% RSLogix 500 project P1.RSS, saved by version 8.10.00.18 %
PROJECT "UNTITLED"    % processor: MicroLogix 1200 %

PROGRAM FILES
  LAD 2 "MAIN"  3 rungs
  LAD 3 "IOS"  5 rungs
  LAD 4 "CONTROL"  11 rungs

DATA FILES
  O0 OUTPUT  4 elements
  I1 INPUT  4 elements
  S2 STATUS  66 elements
  B3 BINARY  1 elements
  T4 TIMER  4 elements
  C5 COUNTER  1 elements
  R6 CONTROL  1 elements
  N7 INTEGER  1 elements

LADDER 2 "MAIN"
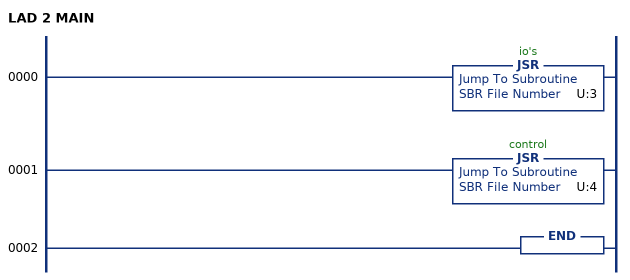
% Rung: 0 %
SOR JSR U:3 EOR
%   U:3  "io's" %
% Rung: 1 %
SOR JSR U:4 EOR
%   U:4  "control" %
% Rung: 2 %
SOR END EOR

LADDER 3 "IOS"
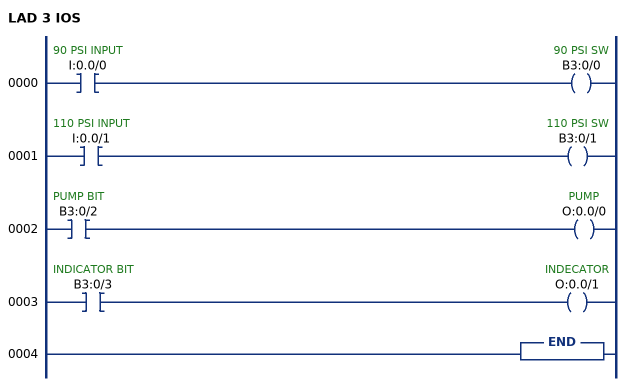
% Rung: 0 %
SOR XIC I:0.0/0 OTE B3:0/0 EOR
%   I:0.0/0  "90 PSI INPUT" %
%   B3:0/0  "90 PSI SW" %
% Rung: 1 %
SOR XIC I:0.0/1 OTE B3:0/1 EOR
%   I:0.0/1  "110 PSI INPUT" %
%   B3:0/1  "110 PSI SW" %
% Rung: 2 %
SOR XIC B3:0/2 OTE O:0.0/0 EOR
%   B3:0/2  "PUMP BIT" %
%   O:0.0/0  "PUMP" %
% Rung: 3 %
SOR XIC B3:0/3 OTE O:0.0/1 EOR
%   B3:0/3  "INDICATOR BIT" %
%   O:0.0/1  "INDECATOR" %
% Rung: 4 %
SOR END EOR

LADDER 4 "CONTROL"
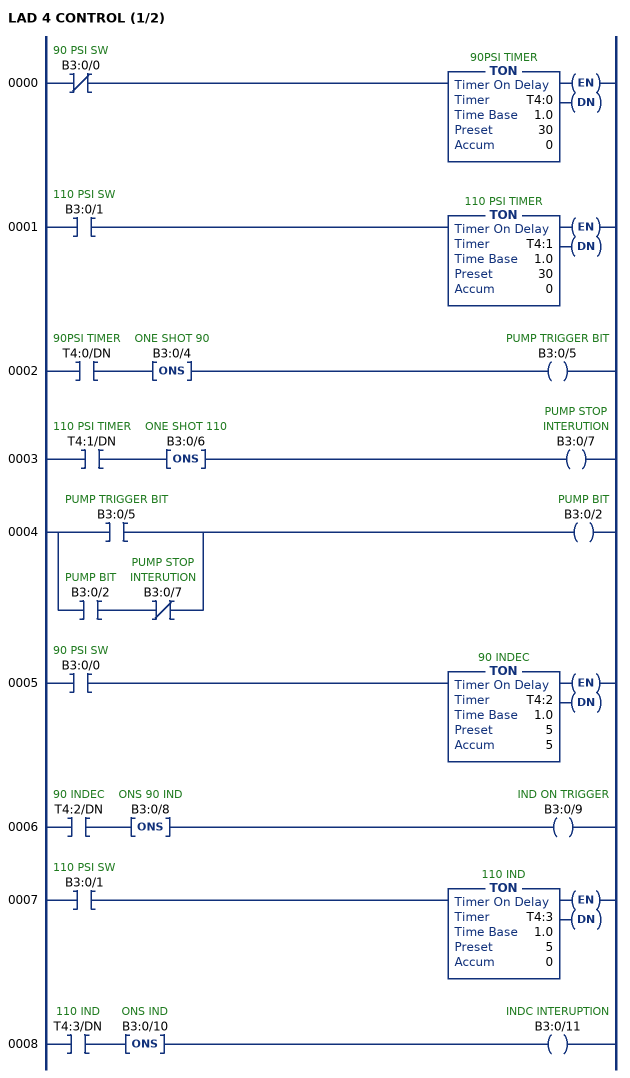
% Rung: 0 %
SOR XIO B3:0/0 TON T4:0 1.0 30 0 EOR
%   B3:0/0  "90 PSI SW" %
%   T4:0  "90PSI TIMER" %
% Rung: 1 %
SOR XIC B3:0/1 TON T4:1 1.0 30 0 EOR
%   B3:0/1  "110 PSI SW" %
%   T4:1  "110 PSI TIMER" %
% Rung: 2 %
SOR XIC T4:0/DN ONS B3:0/4 OTE B3:0/5 EOR
%   T4:0  "90PSI TIMER" %
%   B3:0/4  "ONE SHOT 90" %
%   B3:0/5  "PUMP TRIGGER BIT" %
% Rung: 3 %
SOR XIC T4:1/DN ONS B3:0/6 OTE B3:0/7 EOR
%   T4:1  "110 PSI TIMER" %
%   B3:0/6  "ONE SHOT 110" %
%   B3:0/7  "PUMP STOP INTERUTION" %
% Rung: 4 %
SOR BST XIC B3:0/5 NXB XIC B3:0/2 XIO B3:0/7 BND OTE B3:0/2 EOR
%   B3:0/5  "PUMP TRIGGER BIT" %
%   B3:0/2  "PUMP BIT" %
%   B3:0/7  "PUMP STOP INTERUTION" %
% Rung: 5 %
SOR XIC B3:0/0 TON T4:2 1.0 5 5 EOR
%   B3:0/0  "90 PSI SW" %
%   T4:2  "90 INDEC" %
% Rung: 6 %
SOR XIC T4:2/DN ONS B3:0/8 OTE B3:0/9 EOR
%   T4:2  "90 INDEC" %
%   B3:0/8  "ONS 90 IND" %
%   B3:0/9  "IND ON TRIGGER" %
% Rung: 7 %
SOR XIC B3:0/1 TON T4:3 1.0 5 0 EOR
%   B3:0/1  "110 PSI SW" %
%   T4:3  "110 IND" %
% Rung: 8 %
SOR XIC T4:3/DN ONS B3:0/10 OTE B3:0/11 EOR
%   T4:3  "110 IND" %
%   B3:0/10  "ONS IND" %
%   B3:0/11  "INDC INTERUPTION" %

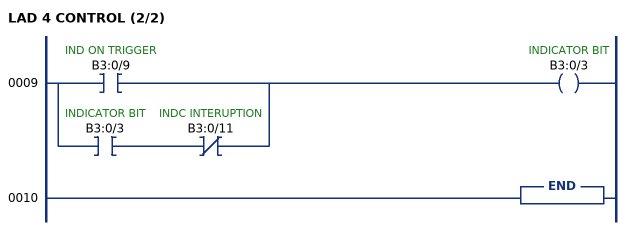
% Rung: 9 %
SOR BST XIC B3:0/9 NXB XIC B3:0/3 XIO B3:0/11 BND OTE B3:0/3 EOR
%   B3:0/9  "IND ON TRIGGER" %
%   B3:0/3  "INDICATOR BIT" %
%   B3:0/11  "INDC INTERUPTION" %
% Rung: 10 %
SOR END EOR

DATA TABLE (non-zero values as saved)
DATA B3
% B3:0 % 0X010D
DATA T4
% .PRE .ACC %
% T4:0 % 30 0
% T4:1 % 30 0
% T4:2 % 5 5
% T4:3 % 5 0
